(* IEC 61131-3 sources: RECIRS/QEMUv8/OpenPLC_v3/webserver/st_files, 24 files *)

(* ---- 7_segment_display.st ---- *)
PROGRAM prog0

VAR
    Rdosc : BOOL;
    Cdigit : INT;
    digit : INT;
    digit0 : INT;
    digit1 : INT;
    digit2 : INT;

    Ycom_digit0 : BOOL;
    Ycom_digit1 : BOOL;
    Ycom_digit2 : BOOL;
    Yseg_a : BOOL;
    Yseg_b : BOOL;
    Yseg_c : BOOL;
    Yseg_d : BOOL;
    Yseg_e : BOOL;
    Yseg_f : BOOL;
    Yseg_g : BOOL;
END_VAR

Rdosc := FALSE;

IF Rdosc THEN
    Rdosc := TRUE;
END_IF;

IF Rdosc THEN
    Cdigit := Cdigit + 1;
    IF Cdigit > 2 THEN
        Cdigit := 0;
    END_IF;
END_IF;

CASE Cdigit OF
    0:
        Ycom_digit0 := TRUE;
        Ycom_digit1 := FALSE;
        Ycom_digit2 := FALSE;
        digit := digit0;
    1:
        Ycom_digit0 := FALSE;
        Ycom_digit1 := TRUE;
        Ycom_digit2 := FALSE;
        digit := digit1;
    2:
        Ycom_digit0 := FALSE;
        Ycom_digit1 := FALSE;
        Ycom_digit2 := TRUE;
        digit := digit2;
END_CASE;

Yseg_a := (digit <> 1) AND (digit <> 4);
Yseg_b := (digit <> 5) AND (digit <> 6);
Yseg_c := (digit <> 2);
Yseg_d := (digit <> 1) AND (digit <> 4) AND (digit <> 7);
Yseg_e := (digit = 0) OR (digit = 2) OR (digit = 6) OR (digit = 8);
Yseg_f := (digit <> 1) AND (digit <> 2) AND (digit <> 3) AND (digit <> 7);
Yseg_g := (digit <> 0) AND (digit <> 1) AND (digit <> 7);

digit0 := 1;
digit1 := 8;
digit2 := 5;

END_PROGRAM

CONFIGURATION Config0

  RESOURCE Res0 ON PLC
    TASK Main(INTERVAL := T#100ms,PRIORITY := 0);
    PROGRAM Inst0 WITH Main : prog0;
  END_RESOURCE
END_CONFIGURATION

(* ---- blank_program.st ---- *)
PROGRAM prog0
  VAR
    var_in : BOOL;
    var_out : BOOL;
  END_VAR

  var_out := var_in;
END_PROGRAM

CONFIGURATION Config0

  RESOURCE Res0 ON PLC
    TASK Main(INTERVAL := T#1ms,PRIORITY := 0);
    PROGRAM Inst0 WITH Main : prog0;
  END_RESOURCE
END_CONFIGURATION

(* ---- brewing_system.st ---- *)
PROGRAM prog0
VAR
    StartButton : BOOL;
    StopButton : BOOL;
    Brewing : BOOL;
    Heating : BOOL;
    Cooling : BOOL;
    Fermenting : BOOL;
    TimerHeat : TON;
    TimerCool : TON;
    TimerFerment : TON;
    StartTrigger : R_TRIG;
    StopTrigger : F_TRIG;
    TempSetPoint : REAL := 65.0;
    _TEMPCurrent : REAL;
    CurrentTemp : REAL := 20.0;
    TempChangeRate : REAL := 0.5;
END_VAR

IF CurrentTemp < TempSetPoint THEN
	StartButton := TRUE;
END_IF;

StartTrigger(CLK := StartButton);
StopTrigger(CLK := StopButton);

IF StartTrigger.Q THEN
    Brewing := TRUE;
    TimerHeat(IN := TRUE, PT := T#1h);
    Heating := TimerHeat.Q;
    IF TimerHeat.Q THEN
        TimerCool(IN := TRUE, PT := T#30m);
        Cooling := TimerCool.Q;
    END_IF;
    IF TimerCool.Q THEN
        TimerFerment(IN := TRUE, PT := T#7d);
        Fermenting := TimerFerment.Q;
    END_IF;
ELSE
    Brewing := FALSE;
    TimerHeat(IN := FALSE);
    TimerCool(IN := FALSE);
    TimerFerment(IN := FALSE);
    Heating := FALSE;
    Cooling := FALSE;
    Fermenting := FALSE;
END_IF;

IF StopTrigger.Q THEN
    Brewing := FALSE;
    Heating := FALSE;
    Cooling := FALSE;
    Fermenting := FALSE;
END_IF;

IF Heating THEN
	_TEMPCurrent := MUL(TempChangeRate, 0.1);
	CurrentTemp := ADD(CurrentTemp, _TEMPCurrent);
ELSIF Cooling THEN
	_TEMPCurrent := MUL(TempChangeRate, 0.1);
	CurrentTemp := SUB(CurrentTemp, _TEMPCurrent);
END_IF;

END_PROGRAM

CONFIGURATION Config0

  RESOURCE Res0 ON PLC
    TASK Main(INTERVAL := T#50ms,PRIORITY := 0);
    PROGRAM Inst0 WITH Main : prog0;
  END_RESOURCE
END_CONFIGURATION

(* ---- car_wash.st ---- *)
PROGRAM prog0
VAR
    StartButton : BOOL := TRUE;
    StopButton : BOOL;
    CarDetected : BOOL;
    Washing : BOOL;
    Rinsing : BOOL;
    Drying : BOOL;
    TimerWash : TON;
    TimerRinse : TON;
    TimerDry : TON;
    StartTrigger : R_TRIG;
    StopTrigger : F_TRIG;
    _TEMP : REAL;
    CarPosition : REAL := 0.0;
    CarSpeed : REAL := 0.5;
    WashPosition : REAL := 2.0;
    RinsePosition : REAL := 4.0;
    DryPosition : REAL := 6.0;
END_VAR

StartTrigger(CLK := StartButton);
StopTrigger(CLK := StopButton);

IF StartTrigger.Q AND CarDetected THEN
    TimerWash(IN := TRUE, PT := T#2m);
    Washing := TimerWash.Q;
    IF TimerWash.Q THEN
        TimerRinse(IN := TRUE, PT := T#1m);
        Rinsing := TimerRinse.Q;
    END_IF;
    IF TimerRinse.Q THEN
        TimerDry(IN := TRUE, PT := T#1m);
        Drying := TimerDry.Q;
    END_IF;
ELSE
    TimerWash(IN := FALSE);
    TimerRinse(IN := FALSE);
    TimerDry(IN := FALSE);
    Washing := FALSE;
    Rinsing := FALSE;
    Drying := FALSE;
END_IF;

IF StopTrigger.Q THEN
    Washing := FALSE;
    Rinsing := FALSE;
    Drying := FALSE;
END_IF;

_TEMP := MUL(CarSpeed, 0.1);
IF Washing THEN
	CarPosition := ADD(CarPosition, _TEMP);
	IF CarPosition >= WashPosition THEN
		Washing := FALSE;
		Rinsing := TRUE;
	END_IF;
END_IF;

IF Rinsing THEN
	CarPosition := ADD(CarPosition, _TEMP);
	IF CarPosition >= RinsePosition THEN
		Rinsing := FALSE;
		Drying := TRUE;
	END_IF;
END_IF;

IF Drying THEN
	CarPosition := ADD(CarPosition, _TEMP);
	IF CarPosition >= DryPosition THEN
		Drying := FALSE;
	END_IF;
END_IF;

END_PROGRAM

CONFIGURATION Config0

  RESOURCE Res0 ON PLC
    TASK Main(INTERVAL := T#50ms,PRIORITY := 0);
    PROGRAM Inst0 WITH Main : prog0;
  END_RESOURCE
END_CONFIGURATION

(* ---- conveyor_belt.st ---- *)
PROGRAM program0
  VAR
    start_button : BOOL;
    stop_button : BOOL;
    emergency_button : BOOL;
    proximity_sensor : BOOL;
    motor_forward : BOOL;
    motor_reverse : BOOL;
    conveyor_running : BOOL := TRUE;
    entity_present : BOOL := FALSE;
    total_types : INT := 1;
    entity_type : INT;
    count : INT := 1;
    timer : BOOL;
    TON0 : TON;
    TOF0 : TOF;
    _TMP_ADD29_OUT : INT;
    _TMP_EQ31_OUT : BOOL;
    _TMP_BOOL_TO_INT33_OUT : INT;
    _TMP_MUL35_OUT : INT;
    _TMP_SUB37_OUT : INT;
    _TMP_INT_TO_STRING39_OUT : STRING;
  END_VAR

  TON0(IN := NOT(timer), PT := T#10ms);
  TOF0(IN := TON0.Q, PT := T#10ms);
  timer := TOF0.Q;
  IF NOT entity_present AND NOT proximity_sensor AND conveyor_running THEN
    entity_present := FALSE;
  END_IF;
  IF proximity_sensor AND conveyor_running THEN
    entity_present := TRUE;
  END_IF;
  entity_type := total_types;
  IF emergency_button THEN
    motor_forward := FALSE;
  END_IF;
  IF NOT conveyor_running THEN
    motor_forward := FALSE;
  END_IF;
  IF emergency_button THEN
    motor_reverse := FALSE;
  END_IF;
  _TMP_ADD29_OUT := ADD(count, 1);
  count := _TMP_ADD29_OUT;
  IF NOT conveyor_running THEN
    motor_reverse := FALSE;
  END_IF;
  IF emergency_button THEN
    conveyor_running := FALSE;
  END_IF;
  IF emergency_button THEN
    entity_present := FALSE;
  END_IF;
  _TMP_EQ31_OUT := EQ(count, 5);
  _TMP_BOOL_TO_INT33_OUT := BOOL_TO_INT(_TMP_EQ31_OUT);
  _TMP_MUL35_OUT := MUL(_TMP_BOOL_TO_INT33_OUT, 4);
  _TMP_SUB37_OUT := SUB(count, _TMP_MUL35_OUT);
  count := _TMP_SUB37_OUT;
  IF start_button AND NOT emergency_button THEN
    conveyor_running := TRUE;
  END_IF;
  IF stop_button AND NOT emergency_button THEN
    conveyor_running := FALSE;
  END_IF;
  _TMP_INT_TO_STRING39_OUT := INT_TO_STRING(entity_type);
END_PROGRAM

CONFIGURATION Config0

  RESOURCE Res0 ON PLC
    TASK task0(INTERVAL := T#100ms,PRIORITY := 0);
    PROGRAM instance0 WITH task0 : program0;
  END_RESOURCE
END_CONFIGURATION

(* ---- elevator.st ---- *)
PROGRAM program0
  VAR
    floor_buttons : ARRAY [1..5] OF BOOL;
    door_sensor : BOOL;
    motor_up : BOOL;
    motor_down : BOOL;
    open_door : BOOL;
    close_door : BOOL;
    current_floor : INT := 1;
    target_floor : INT := 1;
    door_opened : BOOL := FALSE;
    count : INT := 1;
  END_VAR

  IF NOT door_opened THEN
      FOR count := 1 TO 5 DO
          IF floor_buttons[count] THEN
              target_floor := count;
          END_IF;
      END_FOR;
      IF target_floor > current_floor THEN
          motor_up := TRUE;
      ELSIF target_floor < current_floor THEN
          motor_up := FALSE;
          motor_down := TRUE;
      ELSE
          motor_up := FALSE;
          motor_down := FALSE;
      END_IF;
      IF target_floor = current_floor THEN
          motor_up := FALSE;
          motor_down := FALSE;
          open_door := TRUE;
          door_opened := TRUE;
      END_IF;
  ELSE
      IF NOT door_sensor THEN
          close_door := TRUE;
      ELSE
          close_door := FALSE;
          open_door := FALSE;
          door_opened := FALSE;
          current_floor := target_floor;
      END_IF;
  END_IF;
END_PROGRAM

CONFIGURATION Config0

  RESOURCE Res0 ON PLC
    TASK task0(INTERVAL := T#1ms,PRIORITY := 0);
    PROGRAM instance0 WITH task0 : program0;
  END_RESOURCE
END_CONFIGURATION

(* ---- energy_manage.st ---- *)
PROGRAM prog0
VAR
    PeakHours : BOOL;
    NonPeakHours : BOOL;
    EnergyConsumption : REAL := 0.0;
    MaxConsumption : REAL := 1000.0;
    LoadShedding : BOOL;
    Timer : TON;
    _TEMP : REAL;
    EnergyGeneration : REAL := 500.0;
    EnergyUsage : REAL := 600.0;
END_VAR

IF PeakHours THEN
    IF EnergyConsumption > MaxConsumption THEN
        LoadShedding := TRUE;
        Timer(IN := TRUE, PT := T#30m);
    ELSE
        LoadShedding := FALSE;
        Timer(IN := FALSE);
    END_IF;
ELSE
    LoadShedding := FALSE;
    Timer(IN := FALSE);
END_IF;

IF Timer.Q THEN
	LoadShedding := FALSE;
END_IF;

IF LoadShedding THEN
	_TEMP := MUL(EnergyUsage, 0.1);
	EnergyConsumption := SUB(EnergyConsumption, _TEMP);
ELSE
	_TEMP := MUL(EnergyGeneration, 0.1);
	EnergyConsumption := ADD(EnergyConsumption, _TEMP);
END_IF;

END_PROGRAM

CONFIGURATION Config0

  RESOURCE Res0 ON PLC
    TASK Main(INTERVAL := T#50ms,PRIORITY := 0);
    PROGRAM Inst0 WITH Main : prog0;
  END_RESOURCE
END_CONFIGURATION

(* ---- gate_controller.st ---- *)
PROGRAM Gate_Controller
  VAR
    Start_Loop : BOOL := False;
    one_hour : TIME := T#1h;
    One_Hour_Timer : TON;
    Gate_Open : BOOL := False;
  END_VAR
  VAR_OUTPUT
    Close_Gate_Inst : BOOL := False;
  END_VAR
  VAR_INPUT
    Sensed_Car : BOOL := False;
    Sensed_Car_Inst : BOOL := False;
    Sensed_App : BOOL := False;
    Mobile_Inst : BOOL := False;
    Auth : STRING;
  END_VAR
  VAR
    my_defined_str : STRING := '"1234"';
  END_VAR

  One_Hour_Timer(IN := NOT(Start_Loop), PT := one_hour);

  IF One_Hour_Timer.Q THEN
    IF Gate_Open THEN
      Close_Gate_Inst := True;
      Gate_Open := False;
    END_IF;
  END_IF;

  IF Sensed_App THEN
    IF EQ(Auth, my_defined_str) THEN
      Close_Gate_Inst := XOR(Mobile_Inst, Gate_Open);
      Gate_Open := Mobile_Inst;
    END_IF;
  END_IF;

  IF Sensed_Car THEN
    IF EQ(Auth, my_defined_str) THEN
      Close_Gate_Inst := XOR(Sensed_Car_Inst, Gate_Open);
      Gate_Open := Sensed_Car_Inst;
    END_IF;
  END_IF;

  Start_Loop := One_Hour_Timer.Q;
END_PROGRAM

CONFIGURATION Config0

  RESOURCE Res0 ON PLC
    TASK task0(INTERVAL := T#20ms,PRIORITY := 0);
    PROGRAM instance0 WITH task0 : Gate_Controller;
  END_RESOURCE
END_CONFIGURATION

(* ---- greenhouse_climate_ctrl.st ---- *)
PROGRAM prog0
VAR
    TempSetPoint : REAL := 22.0;
    HumiditySetPoint : REAL := 60.0;
    CurrentTemp : REAL := 20.0;
    CurrentHumidity : REAL := 55.0;
    HeaterOn : BOOL;
    CoolerOn : BOOL;
    HumidifierOn : BOOL;
    DehumidifierOn : BOOL;
    VentilationOn : BOOL;
    PIDTemp : PID;
    PIDHumidity : PID;
    _TEMP_HEAT : REAL;
    _TEMP_HUMID : REAL;
    TempChangeRate : REAL := 0.1;
    HumidityChangeRate : REAL := 0.2;
END_VAR

PIDTemp(KP := 2.0, TR := 0.5, TD := 0.1, SP := TempSetPoint, PV := CurrentTemp);
PIDHumidity(KP := 1.5, TR := 0.3, TD := 0.1, SP := HumiditySetPoint, PV := CurrentHumidity);

IF PIDTemp.XOUT > 0.0 THEN
    HeaterOn := TRUE;
    CoolerOn := FALSE;
ELSE
    HeaterOn := FALSE;
    CoolerOn := TRUE;
END_IF;

IF PIDHumidity.XOUT > 0.0 THEN
    HumidifierOn := TRUE;
    DehumidifierOn := FALSE;
ELSE
    HumidifierOn := FALSE;
    DehumidifierOn := FALSE;
END_IF;

IF (CurrentTemp > TempSetPoint + 2.0) OR (CurrentHumidity > HumiditySetPoint + 10.0) THEN
    VentilationOn := TRUE;
ELSE
    VentilationOn := FALSE;
END_IF;

IF HeaterOn THEN
	_TEMP_HEAT := MUL(TempChangeRate, 0.1);
	CurrentTemp := ADD(CurrentTemp, _TEMP_HEAT);
ELSIF CoolerOn THEN
	_TEMP_HEAT := MUL(TempChangeRate, 0.1);
	CurrentTemp := SUB(CurrentTemp, _TEMP_HEAT);
END_IF;

IF HumidifierOn THEN
	_TEMP_HUMID := MUL(HumidityChangeRate, 0.1);
	CurrentHumidity := ADD(CurrentHumidity, _TEMP_HUMID);
ELSIF DehumidifierOn THEN
	_TEMP_HUMID := MUL(HumidityChangeRate, 0.1);
	CurrentHumidity := SUB(CurrentHumidity, _TEMP_HUMID);
END_IF;

END_PROGRAM

CONFIGURATION Config0

  RESOURCE Res0 ON PLC
    TASK Main(INTERVAL := T#50ms,PRIORITY := 0);
    PROGRAM Inst0 WITH Main : prog0;
  END_RESOURCE
END_CONFIGURATION

(* ---- hvac.st ---- *)
PROGRAM program0
  VAR
    Heater_enable AT %IX0.1 : BOOL;
  END_VAR
  VAR
    Heater_power : REAL := 0.0;
    Heater_prop : REAL := 0.3;
    Heater_delay : TIME := T#1s;
  END_VAR
  VAR
    Cooler_enable AT %IX0.2 : BOOL;
  END_VAR
  VAR
    Cooler_power : REAL := 0.0;
    Cooler_prop : REAL := -0.1;
    Cooler_delay : TIME := T#1s;
    Fan_enable : BOOL;
    Fan_power : REAL := 0.0;
    Fan_prop : REAL := 0.2;
  END_VAR
  VAR_EXTERNAL
    temperature : REAL;
    temperature_setpoint : REAL;
  END_VAR
  VAR
    temperature_devi : REAL := 0.1;
    Temperature_MIN : REAL := 0.0;
    Temperature_MAX : REAL := 100.0;
    inner_temperature : REAL := 19.0;
    outer_temperature : REAL := 19.0;
    inout_temperature_prop : REAL := 0.001;
  END_VAR
  VAR_EXTERNAL
    humidity : REAL;
  END_VAR
  VAR
    inner_humidity : REAL := 0.45;
    outer_humidity : REAL := 0.35;
  END_VAR
  VAR_EXTERNAL
    humidity_setpoint : REAL;
  END_VAR
  VAR
    humidity_devi : REAL := 0.01;
    humidity_MIN : REAL := 0.0;
    humidity_MAX : REAL := 1.0;
    inout_humidity_prop : REAL := 0.001;
  END_VAR
  VAR_EXTERNAL
    PID_enable : BOOL;
    PID1_enable : BOOL;
    PID_out : REAL;
    PID1_out : REAL;
  END_VAR
  VAR
    PID_zero : REAL := 0.0;
    TON0 : TON;
    TON1 : TON;
    _TMP_ADD87_OUT : REAL;
    _TMP_GT84_OUT : BOOL;
    _TMP_SUB90_OUT : REAL;
    _TMP_LT89_OUT : BOOL;
    _TMP_LIMIT52_OUT : REAL;
    _TMP_LIMIT124_OUT : REAL;
    _TMP_GT72_OUT : BOOL;
    _TMP_EQ65_OUT : BOOL;
    _TMP_LT71_OUT : BOOL;
    _TMP_ADD33_OUT : REAL;
    _TMP_LT29_OUT : BOOL;
    _TMP_SUB38_OUT : REAL;
    _TMP_GT35_OUT : BOOL;
    _TMP_AND91_OUT : BOOL;
    _TMP_MUL6_OUT : REAL;
    _TMP_MUL9_OUT : REAL;
    _TMP_GT93_OUT : BOOL;
    _TMP_BOOL_TO_REAL47_OUT : REAL;
    _TMP_MUL48_OUT : REAL;
    _TMP_ADD49_OUT : REAL;
    _TMP_LT73_OUT : BOOL;
    _TMP_BOOL_TO_REAL58_OUT : REAL;
    _TMP_MUL59_OUT : REAL;
    _TMP_SUB61_OUT : REAL;
    _TMP_BOOL_TO_REAL41_OUT : REAL;
    _TMP_MUL17_OUT : REAL;
    _TMP_ADD40_OUT : REAL;
    _TMP_BOOL_TO_REAL12_OUT : REAL;
    _TMP_MUL23_OUT : REAL;
    _TMP_SUB22_OUT : REAL;
    _TMP_GT108_OUT : BOOL;
    _TMP_BOOL_TO_REAL74_OUT : REAL;
    _TMP_MUL94_OUT : REAL;
    _TMP_ADD96_OUT : REAL;
    _TMP_EQ112_OUT : BOOL;
    _TMP_LT105_OUT : BOOL;
    _TMP_BOOL_TO_REAL100_OUT : REAL;
    _TMP_MUL101_OUT : REAL;
    _TMP_SUB102_OUT : REAL;
    _TMP_MUL118_OUT : REAL;
    _TMP_ADD120_OUT : REAL;
    _TMP_SUB139_OUT : REAL;
    _TMP_LT134_OUT : BOOL;
    _TMP_ADD133_OUT : REAL;
    _TMP_GT131_OUT : BOOL;
    _TMP_ADD147_OUT : REAL;
    _TMP_LT143_OUT : BOOL;
    _TMP_SUB151_OUT : REAL;
    _TMP_GT155_OUT : BOOL;
    _TMP_AND152_OUT : BOOL;
  END_VAR

  _TMP_ADD87_OUT := ADD(temperature_setpoint, temperature_devi);
  _TMP_GT84_OUT := GT(temperature, _TMP_ADD87_OUT);
  _TMP_SUB90_OUT := SUB(temperature_setpoint, temperature_devi);
  _TMP_LT89_OUT := LT(temperature, _TMP_SUB90_OUT);
  IF _TMP_GT84_OUT OR _TMP_LT89_OUT THEN
    PID_enable := TRUE; (*set*)
  END_IF;
  _TMP_LIMIT52_OUT := LIMIT(Temperature_MIN, inner_temperature, Temperature_MAX);
  temperature := _TMP_LIMIT52_OUT;
  IF NOT(PID_enable) THEN
    Heater_enable := FALSE; (*reset*)
  END_IF;
  IF NOT(PID_enable) THEN
    Cooler_enable := FALSE; (*reset*)
  END_IF;
  _TMP_LIMIT124_OUT := LIMIT(humidity_MIN, inner_humidity, humidity_MAX);
  humidity := _TMP_LIMIT124_OUT;
  _TMP_GT72_OUT := GT(PID_out, PID_zero);
  IF _TMP_GT72_OUT THEN
    Heater_enable := TRUE; (*set*)
  END_IF;
  _TMP_EQ65_OUT := EQ(PID_out, PID_zero);
  _TMP_LT71_OUT := LT(PID_out, PID_zero);
  IF _TMP_EQ65_OUT OR _TMP_LT71_OUT THEN
    Heater_enable := FALSE; (*reset*)
  END_IF;
  _TMP_ADD33_OUT := ADD(temperature_setpoint, temperature_devi);
  _TMP_LT29_OUT := LT(temperature, _TMP_ADD33_OUT);
  _TMP_SUB38_OUT := SUB(temperature_setpoint, temperature_devi);
  _TMP_GT35_OUT := GT(temperature, _TMP_SUB38_OUT);
  _TMP_AND91_OUT := AND(_TMP_LT29_OUT, _TMP_GT35_OUT);
  IF _TMP_AND91_OUT THEN
    PID_enable := FALSE; (*reset*)
  END_IF;
  IF _TMP_EQ65_OUT OR _TMP_GT72_OUT THEN
    Cooler_enable := FALSE; (*reset*)
  END_IF;
  IF _TMP_LT71_OUT THEN
    Cooler_enable := TRUE; (*set*)
  END_IF;
  _TMP_MUL6_OUT := MUL(PID_out, Heater_prop);
  Heater_power := _TMP_MUL6_OUT;
  _TMP_MUL9_OUT := MUL(PID_out, Cooler_prop);
  Cooler_power := _TMP_MUL9_OUT;
  _TMP_GT93_OUT := GT(outer_temperature, inner_temperature);
  _TMP_BOOL_TO_REAL47_OUT := BOOL_TO_REAL(_TMP_GT93_OUT);
  _TMP_MUL48_OUT := MUL(_TMP_BOOL_TO_REAL47_OUT, inout_temperature_prop);
  _TMP_ADD49_OUT := ADD(_TMP_MUL48_OUT, inner_temperature);
  inner_temperature := _TMP_ADD49_OUT;
  _TMP_LT73_OUT := LT(outer_temperature, inner_temperature);
  _TMP_BOOL_TO_REAL58_OUT := BOOL_TO_REAL(_TMP_LT73_OUT);
  _TMP_MUL59_OUT := MUL(_TMP_BOOL_TO_REAL58_OUT, inout_temperature_prop);
  _TMP_SUB61_OUT := SUB(inner_temperature, _TMP_MUL59_OUT);
  inner_temperature := _TMP_SUB61_OUT;
  TON0(IN := Heater_enable, PT := Heater_delay);
  _TMP_BOOL_TO_REAL41_OUT := BOOL_TO_REAL(TON0.Q);
  _TMP_MUL17_OUT := MUL(_TMP_BOOL_TO_REAL41_OUT, Heater_power);
  _TMP_ADD40_OUT := ADD(_TMP_MUL17_OUT, inner_temperature);
  inner_temperature := _TMP_ADD40_OUT;
  TON1(IN := Cooler_enable, PT := Cooler_delay);
  _TMP_BOOL_TO_REAL12_OUT := BOOL_TO_REAL(TON1.Q);
  _TMP_MUL23_OUT := MUL(_TMP_BOOL_TO_REAL12_OUT, Cooler_power);
  _TMP_SUB22_OUT := SUB(inner_temperature, _TMP_MUL23_OUT);
  inner_temperature := _TMP_SUB22_OUT;
  _TMP_GT108_OUT := GT(outer_humidity, inner_humidity);
  _TMP_BOOL_TO_REAL74_OUT := BOOL_TO_REAL(_TMP_GT108_OUT);
  _TMP_MUL94_OUT := MUL(_TMP_BOOL_TO_REAL74_OUT, inout_humidity_prop);
  _TMP_ADD96_OUT := ADD(_TMP_MUL94_OUT, inner_humidity);
  inner_humidity := _TMP_ADD96_OUT;
  _TMP_EQ112_OUT := EQ(PID1_out, PID_zero);
  IF _TMP_EQ112_OUT THEN
    Fan_enable := FALSE; (*reset*)
  END_IF;
  IF PID1_enable THEN
    Fan_enable := TRUE; (*set*)
  END_IF;
  _TMP_LT105_OUT := LT(outer_humidity, inner_humidity);
  _TMP_BOOL_TO_REAL100_OUT := BOOL_TO_REAL(_TMP_LT105_OUT);
  _TMP_MUL101_OUT := MUL(_TMP_BOOL_TO_REAL100_OUT, inout_humidity_prop);
  _TMP_SUB102_OUT := SUB(inner_humidity, _TMP_MUL101_OUT);
  inner_humidity := _TMP_SUB102_OUT;
  _TMP_MUL118_OUT := MUL(PID1_out, Fan_prop);
  Fan_power := _TMP_MUL118_OUT;
  _TMP_ADD120_OUT := ADD(inner_humidity, Fan_power);
  inner_humidity := _TMP_ADD120_OUT;
  _TMP_SUB139_OUT := SUB(humidity_setpoint, humidity_devi);
  _TMP_LT134_OUT := LT(temperature, _TMP_SUB139_OUT);
  _TMP_ADD133_OUT := ADD(humidity_setpoint, humidity_devi);
  _TMP_GT131_OUT := GT(humidity, _TMP_ADD133_OUT);
  IF _TMP_GT131_OUT OR _TMP_LT134_OUT THEN
    PID1_enable := TRUE; (*set*)
  END_IF;
  _TMP_ADD147_OUT := ADD(humidity_setpoint, humidity_devi);
  _TMP_LT143_OUT := LT(humidity, _TMP_ADD147_OUT);
  _TMP_SUB151_OUT := SUB(humidity_setpoint, humidity_devi);
  _TMP_GT155_OUT := GT(humidity, _TMP_SUB151_OUT);
  _TMP_AND152_OUT := AND(_TMP_LT143_OUT, _TMP_GT155_OUT);
  IF _TMP_AND152_OUT THEN
    PID1_enable := FALSE; (*reset*)
  END_IF;
END_PROGRAM

PROGRAM program1
  VAR
    PID0 : PID;
  END_VAR
  VAR_EXTERNAL
    PID_enable : BOOL;
  END_VAR
  VAR
    PID_X0 : REAL;
    PID_KP : REAL := -0.05;
    PID_TR : REAL := 10.0;
    PID_TD : REAL := 40.0;
    PID_CYCLE : TIME := T#10ms;
  END_VAR
  VAR_EXTERNAL
    temperature : REAL;
    PID_out : REAL;
    temperature_setpoint : REAL;
  END_VAR

  PID0(AUTO := PID_enable, PV := temperature, SP := temperature_setpoint, KP := PID_KP, TR := PID_TR, TD := PID_TD, CYCLE := PID_CYCLE);
  PID_out := PID0.XOUT;
END_PROGRAM

PROGRAM program2
  VAR
    PID1 : PID;
  END_VAR
  VAR_EXTERNAL
    PID1_enable : BOOL;
  END_VAR
  VAR
    PID1_X0 : REAL;
    PID1_KP : REAL := -0.01;
    PID1_TR : REAL := 5.0;
    PID1_TD : REAL := 20.0;
    PID1_CYCLE : TIME := T#10ms;
  END_VAR
  VAR_EXTERNAL
    humidity : REAL;
    PID1_out : REAL;
    humidity_setpoint : REAL;
  END_VAR

  PID1(AUTO := PID1_enable, PV := humidity, SP := humidity_setpoint, KP := PID1_KP, TR := PID1_TR, TD := PID1_TD, CYCLE := PID1_CYCLE);
  PID1_out := PID1.XOUT;
END_PROGRAM

CONFIGURATION Config0

  RESOURCE Res0 ON PLC
    VAR_GLOBAL
      temperature AT %MD0 : REAL := 0.0;
      humidity AT %MD4 : REAL := 0.0;
      PID_out AT %MD8 : REAL := 0.0;
      PID1_out AT %MD12 : REAL := 0.0;
      PID_enable : BOOL := 1;
      PID1_enable : BOOL := 1;
      temperature_setpoint AT %MD16 : REAL := 24.0;
      humidity_setpoint AT %MD20 : REAL := 0.35;
    END_VAR
    TASK task0(INTERVAL := T#10ms,PRIORITY := 0);
    TASK task2(INTERVAL := T#10ms,PRIORITY := 0);
    TASK task1(INTERVAL := T#10ms,PRIORITY := 0);
    PROGRAM instance0 WITH task0 : program0;
    PROGRAM instance2 WITH task2 : program2;
    PROGRAM instance1 WITH task1 : program1;
  END_RESOURCE
END_CONFIGURATION

(* ---- irrigation_system.st ---- *)
PROGRAM prog0
VAR
    SoilMoisture : REAL := 40.0;
    MoistureSetPoint : REAL := 50.0;
    MoistureUpperLimit : REAL := 60.0;
    MoistureLowerLimit : REAL := 30.0;
    IrrigationOn : BOOL;
    IrrigationAddRate : REAL := 5.0;
    Timer : TON;
    MoistureDecayRate : REAL := 0.5;
END_VAR

IF SoilMoisture < MoistureLowerLimit THEN
    IrrigationOn := TRUE;
    Timer(IN := TRUE, PT := T#30m);
ELSE
    IrrigationOn := FALSE;
    Timer(IN := FALSE);
END_IF;

IF Timer.Q THEN
    IrrigationOn := FALSE;
END_IF;

IF IrrigationOn THEN
	SoilMoisture := ADD(SoilMoisture, IrrigationAddRate);
END_IF;

SoilMoisture := SUB(SoilMoisture, MoistureDecayRate);

END_PROGRAM

CONFIGURATION Config0

  RESOURCE Res0 ON PLC
    TASK Main(INTERVAL := T#1s,PRIORITY := 0);
    PROGRAM Inst0 WITH Main : prog0;
  END_RESOURCE
END_CONFIGURATION

(* ---- lighting_system.st ---- *)
PROGRAM prog0
VAR
    MotionDetected : BOOL;
    LightLevel : REAL;
    LightThreshold : REAL := 300.0;
    LightOn : BOOL;
    Timer : TON;
    MotionTrigger : R_TRIG;
    _TEMP : REAL;
    LightDecayRate : REAL := 10.0;
END_VAR

MotionTrigger(CLK := MotionDetected);

IF MotionTrigger.Q THEN
    LightOn := TRUE;
    Timer(IN := TRUE, PT := T#5m);
ELSE
    Timer(IN := FALSE);
END_IF;

IF Timer.Q THEN
    LightOn := FALSE;
END_IF;

IF LightLevel < LightThreshold THEN
    LightOn := TRUE;
ELSE
    LightOn := FALSE;
END_IF;

IF LightOn THEN
	_TEMP := MUL(LightDecayRate, 0.1);
	LightLevel := ADD(LightLevel, _TEMP);
ELSE
	_TEMP := MUL(LightDecayRate, 0.1);
	LightLevel := SUB(LightLevel, _TEMP);
END_IF;

END_PROGRAM

CONFIGURATION Config0

  RESOURCE Res0 ON PLC
    TASK Main(INTERVAL := T#50ms,PRIORITY := 0);
    PROGRAM Inst0 WITH Main : prog0;
  END_RESOURCE
END_CONFIGURATION

(* ---- packaging_system.st ---- *)
PROGRAM prog0
VAR
    StartButton : BOOL := TRUE;
    StopButton : BOOL;
    ConveyorRunning : BOOL;
    PackageDetected : BOOL;
    PackageCount : INT := 0;
    MaxPackages : INT := 100;
    SealerOn : BOOL;
    EjectorOn : BOOL;
    TimerSealer : TON;
    TimerEjector : TON;
    StartTrigger : R_TRIG;
    StopTrigger : F_TRIG;
    ConveyorSpeed : REAL := 1.0;
    ConveyorPosition : REAL := 0.0;
    PackagePositon : REAL := 0.0;
	PackageLength : REAL := 0.5;
	_TEMPPOS : REAL;
END_VAR

StartTrigger(CLK := StartButton);
StopTrigger(CLK := StopButton);

IF StartButton THEN
    ConveyorRunning := TRUE;
ELSIF StopButton THEN
    ConveyorRunning := FALSE;
END_IF;

IF ConveyorRunning THEN
	_TEMPPOS := MUL(ConveyorSpeed, 0.1);
	ConveyorPosition := ADD(ConveyorPosition, _TEMPPOS);
	IF ConveyorPosition >= PackagePositon + PackageLength THEN
		PackageDetected := TRUE;
		PackagePositon := ConveyorPosition;
	ELSE
		PackageDetected := FALSE;
	END_IF;
ELSE
	PackageDetected := FALSE;
END_IF;

IF ConveyorRunning AND PackageDetected THEN
    PackageCount := PackageCount + 1;
    TimerSealer(IN := TRUE, PT := T#5s);
    SealerOn := TimerSealer.Q;
    IF TimerSealer.Q THEN
		TimerEjector(IN := TRUE, PT := T#2s);
		EjectorOn := TimerEjector.Q;
	END_IF;
    IF PackageCount >= MaxPackages THEN
        ConveyorRunning := FALSE;
    END_IF;
ELSE
    TimerSealer(IN := FALSE);
    TimerEjector(IN := FALSE);
    SealerOn := FALSE;
    EjectorOn := FALSE;
END_IF;
END_PROGRAM

CONFIGURATION Config0

  RESOURCE Res0 ON PLC
    TASK Main(INTERVAL := T#50ms,PRIORITY := 0);
    PROGRAM Inst0 WITH Main : prog0;
  END_RESOURCE
END_CONFIGURATION

(* ---- painting_system.st ---- *)
PROGRAM prog0
VAR
    StartButton : BOOL;
    StopButton : BOOL;
    Painting : BOOL;
    PaintLevel : REAL := 0.0;
    PaintThreshold : REAL := 10.0;
    _TEMPPAINT : REAL;
    RefillPaint : BOOL;
    Timer : TON;
    StartTrigger : R_TRIG;
    StopTrigger : F_TRIG;
    PaintUsageRate : REAL := 1.0;
END_VAR

StartTrigger(CLK := StartButton);
StopTrigger(CLK := StopButton);

IF StartTrigger.Q THEN
    Painting := TRUE;
    Timer(IN := TRUE, PT := T#10m);
ELSIF StopTrigger.Q THEN
    Painting := FALSE;
    Timer(IN := FALSE);
END_IF;

IF PaintLevel < PaintThreshold THEN
	StopButton := FALSE;
	StartButton := TRUE;
ELSIF PaintLevel = 100.0 THEN
	StopButton := TRUE;
	StartButton := FALSE;
END_IF;

IF Timer.Q THEN
    Painting := FALSE;
END_IF;

IF Painting THEN
	_TEMPPAINT := MUL(PaintUsageRate, 0.5);
	PaintLevel := ADD(PaintLevel, _TEMPPAINT);
ELSE
	_TEMPPAINT := MUL(PaintUsageRate, 0.1);
	PaintLevel := SUB(PaintLevel, _TEMPPAINT);
END_IF;

END_PROGRAM

CONFIGURATION Config0

  RESOURCE Res0 ON PLC
    TASK Main(INTERVAL := T#50ms,PRIORITY := 0);
    PROGRAM Inst0 WITH Main : prog0;
  END_RESOURCE
END_CONFIGURATION

(* ---- PWM.st ---- *)
PROGRAM program0
  VAR
    level : DINT;
    count : INT := 1;
    input_analog : REAL;
    input_analog_MIN : REAL := 0.0;
    input_analog_MAX : REAL := 3.3;
    input_analog_local : REAL := 0.0;
    _TMP_INT_TO_REAL42_OUT : REAL;
    _TMP_SIN47_OUT : REAL;
    _TMP_ADD48_OUT : REAL;
    _TMP_MUL43_OUT : REAL;
    _TMP_LIMIT35_OUT : INT;
    _TMP_LIMIT31_OUT : REAL;
    _TMP_DIV23_OUT : REAL;
    _TMP_MUL25_OUT : REAL;
    _TMP_REAL_TO_DINT27_OUT : DINT;
    _TMP_EQ29_OUT : BOOL;
    _TMP_BOOL_TO_INT44_OUT : INT;
    _TMP_MUL45_OUT : INT;
    _TMP_SUB46_OUT : INT;
    _TMP_ADD19_OUT : INT;
  END_VAR

  _TMP_INT_TO_REAL42_OUT := INT_TO_REAL(count);
  _TMP_SIN47_OUT := SIN(_TMP_INT_TO_REAL42_OUT);
  _TMP_ADD48_OUT := ADD(_TMP_SIN47_OUT, 1.0);
  _TMP_MUL43_OUT := MUL(_TMP_ADD48_OUT, 1.65);
  input_analog := _TMP_MUL43_OUT;
  _TMP_LIMIT35_OUT := LIMIT(1, count, 200);
  count := _TMP_LIMIT35_OUT;
  _TMP_LIMIT31_OUT := LIMIT(input_analog_MIN, input_analog, input_analog_MAX);
  input_analog_local := _TMP_LIMIT31_OUT;
  _TMP_DIV23_OUT := DIV(input_analog_local, input_analog_MAX);
  _TMP_MUL25_OUT := MUL(_TMP_DIV23_OUT, 65535.0);
  _TMP_REAL_TO_DINT27_OUT := REAL_TO_DINT(_TMP_MUL25_OUT);
  level := _TMP_REAL_TO_DINT27_OUT;
  _TMP_EQ29_OUT := EQ(count, 200);
  _TMP_BOOL_TO_INT44_OUT := BOOL_TO_INT(_TMP_EQ29_OUT);
  _TMP_MUL45_OUT := MUL(_TMP_BOOL_TO_INT44_OUT, 200);
  _TMP_SUB46_OUT := SUB(count, _TMP_MUL45_OUT);
  count := _TMP_SUB46_OUT;
  _TMP_ADD19_OUT := ADD(count, 1);
  count := _TMP_ADD19_OUT;
END_PROGRAM

CONFIGURATION Config0

  RESOURCE Res0 ON PLC
    TASK task0(INTERVAL := T#20ms,PRIORITY := 0);
    PROGRAM instance0 WITH task0 : program0;
  END_RESOURCE
END_CONFIGURATION

(* ---- robot_arm_ctrl.st ---- *)
PROGRAM prog0
VAR
    StartButton : BOOL := TRUE;
    StopButton : BOOL;
    ArmPosition : REAL := 0.0;
    TargetPosition : REAL := 100.0;
    ArmMoving : BOOL;
    ArmSpeed : REAL := 10.0;
    Timer : TON;
    StartTrigger : R_TRIG;
    StopTrigger : F_TRIG;
    ArmAcceleration : REAL := 1.0;
    ArmVelocity : REAL := 0.0;
    _TempArmPosition : REAL;
    _TempTimer : REAL;
END_VAR

StartTrigger(CLK := StartButton);
StopTrigger(CLK := StopButton);

IF StartTrigger.Q THEN
    ArmMoving := TRUE;
    Timer(IN := TRUE, PT := T#10s);
ELSIF StopTrigger.Q THEN
    ArmMoving := FALSE;
    Timer(IN := FALSE);
END_IF;

IF ArmMoving THEN
    IF ArmPosition < TargetPosition THEN
		_TempTimer := TIME_TO_REAL(Timer.ET);
		_TempArmPosition := MUL(ArmSpeed, _TempTimer);
        ArmPosition := ADD(ArmPosition, _TempArmPosition);
    ELSE
        ArmMoving := FALSE;
    END_IF;
END_IF;
END_PROGRAM

CONFIGURATION Config0

  RESOURCE Res0 ON PLC
    TASK Main(INTERVAL := T#50ms,PRIORITY := 0);
    PROGRAM Inst0 WITH Main : prog0;
  END_RESOURCE
END_CONFIGURATION

(* ---- solar_power_manage.st ---- *)
PROGRAM prog0
VAR
    SolarPanelOutput : REAL := 500.0;
    BatteryLevel : REAL := 50.0;
    GridSupply : REAL := 0.0;
    LoadDemand : REAL := 600.0;
    BatteryCharging : BOOL;
    GridSupplyOn : BOOL;
    Timer : TON;
    _TEMP : REAL;
    BatteryDischargeRate : REAL := 10.0;
END_VAR

IF SolarPanelOutput > LoadDemand THEN
    BatteryCharging := TRUE;
    GridSupplyOn := FALSE;
    Timer(IN := TRUE, PT := T#1h);
ELSE
    BatteryCharging := FALSE;
    Timer(IN := FALSE);
    IF BatteryLevel < 20.0 THEN
        GridSupplyOn := TRUE;
    ELSE
        GridSupplyOn := FALSE;
    END_IF;
END_IF;

IF Timer.Q THEN
	BatteryCharging := FALSE;
END_IF;

IF BatteryCharging THEN
	_TEMP := MUL(BatteryDischargeRate, 0.1);
	BatteryLevel := ADD(BatteryLevel, _TEMP);
ELSE
	_TEMP := MUL(BatteryDischargeRate, 0.1);
	BatteryLevel := SUB(BatteryLevel, _TEMP);
END_IF;
END_PROGRAM

CONFIGURATION Config0

  RESOURCE Res0 ON PLC
    TASK Main(INTERVAL := T#50ms,PRIORITY := 0);
    PROGRAM Inst0 WITH Main : prog0;
  END_RESOURCE
END_CONFIGURATION

(* ---- sorting_system.st ---- *)
PROGRAM prog0
VAR
    StartButton : BOOL;
    StopButton : BOOL;
    ConveyorRunning : BOOL;
    ItemDetected : BOOL;
    ItemType : INT;
    SortBin1 : BOOL;
    SortBin2 : BOOL;
    SortBin3 : BOOL;
    Timer : TON;
    StartTrigger : R_TRIG;
    StopTrigger : F_TRIG;
    _TEMPPOS : REAL;
    ConveyorSpeed : REAL := 1.0;
    ConveyorPosition : REAL := 0.0;
    ItemPosition : REAL := 0.0;
    Bin1Position : REAL := 2.0;
    Bin2Position : REAL := 4.0;
    Bin3Position : REAL := 6.0;
END_VAR

StartTrigger(CLK := StartButton);
StopTrigger(CLK := StopButton);

IF StartTrigger.Q THEN
    ConveyorRunning := TRUE;
ELSIF StopTrigger.Q THEN
    ConveyorRunning := FALSE;
END_IF;

IF ConveyorRunning THEN
	_TEMPPOS := MUL(ConveyorSpeed, 0.1);
	ConveyorPosition := ADD(ConveyorPosition, _TEMPPOS);
	IF ConveyorPosition >= ItemPosition + 1.0 THEN
		ItemDetected := TRUE;
		ItemPosition := ConveyorPosition;
	ELSE
		ItemDetected := FALSE;
	END_IF;
ELSE
	ItemDetected := FALSE;
END_IF;

IF ConveyorRunning AND ItemDetected THEN
    CASE ItemType OF
        1:
			SortBin1 := TRUE;
			Timer(IN := TRUE, PT := T#2s);
        2:
			SortBin2 := TRUE;
			Timer(IN := TRUE, PT := T#2s);
        3:
			SortBin3 := TRUE;
			Timer(IN := TRUE, PT := T#2s);
    ELSE
        SortBin1 := FALSE;
        SortBin2 := FALSE;
        SortBin3 := FALSE;
    END_CASE;
END_IF;

IF Timer.Q THEN
	SortBin1 := FALSE;
	SortBin2 := FALSE;
	SortBin3 := FALSE;
END_IF;

END_PROGRAM

CONFIGURATION Config0

  RESOURCE Res0 ON PLC
    TASK Main(INTERVAL := T#50ms,PRIORITY := 0);
    PROGRAM Inst0 WITH Main : prog0;
  END_RESOURCE
END_CONFIGURATION

(* ---- traffic_light.st ---- *)
PROGRAM Trafic_light
  VAR
    TOF0 : TOF;
    Always_True : BOOL := True;
    Delay_PLC_start_up : BOOL;
    TOF1 : TOF;
    TOF2 : TOF;
  END_VAR
  VAR
    O_LEDRed AT %QX100.0 : BOOL;
    O_LEDOrange AT %QX100.1 : BOOL;
    O_LEDGreen AT %QX100.2 : BOOL;
  END_VAR
  VAR
    No_lamps_active_for_1s : BOOL;
    F_TRIG0 : F_TRIG;
    F_TRIG1 : F_TRIG;
    F_TRIG2 : F_TRIG;
    TON0 : TON;
    SR0 : SR;
    TOF3 : TOF;
    TOF4 : TOF;
    TOF5 : TOF;
    _TMP_OR22_OUT : BOOL;
    _TMP_AND29_OUT : BOOL;
    _TMP_AND33_OUT : BOOL;
    _TMP_AND34_OUT : BOOL;
    _TMP_OR13_OUT : BOOL;
    _TMP_NOT14_OUT : BOOL;
  END_VAR

  TON0(IN := Always_True, PT := T#2s);
  SR0(S1 := TON0.Q);
  Delay_PLC_start_up := SR0.Q1;
  F_TRIG2(CLK := O_LEDOrange);
  _TMP_OR22_OUT := OR(No_lamps_active_for_1s, F_TRIG2.Q);
  TOF0(IN := _TMP_OR22_OUT, PT := T#10s);
  _TMP_AND29_OUT := AND(TOF0.Q, Delay_PLC_start_up);
  O_LEDRed := _TMP_AND29_OUT;
  F_TRIG0(CLK := O_LEDGreen);
  TOF1(IN := F_TRIG0.Q, PT := T#4s);
  _TMP_AND33_OUT := AND(TOF1.Q, Delay_PLC_start_up);
  O_LEDOrange := _TMP_AND33_OUT;
  F_TRIG1(CLK := O_LEDRed);
  TOF2(IN := F_TRIG1.Q, PT := T#10s);
  _TMP_AND34_OUT := AND(TOF2.Q, Delay_PLC_start_up);
  O_LEDGreen := _TMP_AND34_OUT;
  TOF3(IN := O_LEDRed, PT := T#1s);
  TOF4(IN := O_LEDGreen, PT := T#1s);
  TOF5(IN := O_LEDOrange, PT := T#1s);
  _TMP_OR13_OUT := OR(TOF3.Q, TOF4.Q, TOF5.Q);
  _TMP_NOT14_OUT := NOT(_TMP_OR13_OUT);
  No_lamps_active_for_1s := _TMP_NOT14_OUT;
END_PROGRAM

CONFIGURATION Config0

  RESOURCE Res0 ON PLC
    TASK task0(INTERVAL := T#20ms,PRIORITY := 0);
    PROGRAM instance0 WITH task0 : Trafic_light;
  END_RESOURCE
END_CONFIGURATION

(* ---- warehouse_system.st ---- *)
PROGRAM prog0
VAR
    StartButton : BOOL := TRUE;
    StopButton : BOOL;
    ConveyorRunning : BOOL;
    ItemDetected : BOOL;
    StorageLocation : INT;
    ArmMoving : BOOL;
    ArmPosition : REAL;
    TargetPosition : REAL := 0.0;
    Timer : TON;
    StartTrigger : R_TRIG;
    StopTrigger : F_TRIG;
    _TEMPPOS : REAL;
    ConveyorSpeed : REAL := 1.0;
    ConveyorPosition : REAL := 0.0;
    ItemPosition : REAL := 0.0;
END_VAR

StartTrigger(CLK := StartButton);
StopTrigger(CLK := StopButton);

IF StartTrigger.Q THEN
    ConveyorRunning := TRUE;
ELSIF StopTrigger.Q THEN
    ConveyorRunning := FALSE;
END_IF;

IF ConveyorRunning THEN
	_TEMPPOS := MUL(ConveyorSpeed, 0.1);
	ConveyorPosition := ADD(ConveyorPosition, _TEMPPOS);
	IF ConveyorPosition >= ItemPosition + 1.0 THEN
		ItemDetected := TRUE;
		ItemPosition := ConveyorPosition;
	ELSE
		ItemDetected := FALSE;
	END_IF;
ELSE
	ItemDetected := FALSE;
END_IF;

IF ConveyorRunning AND ItemDetected THEN
    CASE StorageLocation OF
        1: TargetPosition := 10.0;
        2: TargetPosition := 20.0;
        3: TargetPosition := 30.0;
    ELSE
        TargetPosition := 0.0;
    END_CASE;
    ArmMoving := TRUE;
    Timer(IN := TRUE, PT := T#5s);
END_IF;

IF ArmMoving THEN
    IF ArmPosition < TargetPosition THEN
        ArmPosition := ArmPosition + 1.0;
    ELSE
        ArmMoving := FALSE;
    END_IF;
END_IF;

IF Timer.Q THEN
	ArmMoving := FALSE;
END_IF;

END_PROGRAM

CONFIGURATION Config0

  RESOURCE Res0 ON PLC
    TASK Main(INTERVAL := T#50ms,PRIORITY := 0);
    PROGRAM Inst0 WITH Main : prog0;
  END_RESOURCE
END_CONFIGURATION

(* ---- watertank.st ---- *)
PROGRAM program0
  VAR
    Valve_in : BOOL;
  END_VAR
  VAR_INPUT
    Valve_in_input : BOOL;
  END_VAR
  VAR
    Valve_out : BOOL;
  END_VAR
  VAR_INPUT
    Valve_out_input : BOOL;
  END_VAR
  VAR_EXTERNAL
    water_height : REAL;
  END_VAR
  VAR
    water_heigh_MIN : REAL := 0.0;
    water_height_MAX : REAL := 100.0;
    inner_water_height : REAL := 100.0;
  END_VAR
  VAR_EXTERNAL
    Valve_in_rate : REAL;
  END_VAR
  VAR
    Valve_in_rate_MIN : REAL := 0.0;
    Valve_in_rate_MAX : REAL := 3.0;
    inner_Valve_in_rate : REAL := 0.0;
    Valve_out_rate : REAL := 0.3;
    _TMP_BOOL_TO_REAL41_OUT : REAL;
    _TMP_MUL17_OUT : REAL;
    _TMP_ADD40_OUT : REAL;
    _TMP_BOOL_TO_REAL12_OUT : REAL;
    _TMP_MUL23_OUT : REAL;
    _TMP_SQRT51_OUT : REAL;
    _TMP_MUL27_OUT : REAL;
    _TMP_SUB22_OUT : REAL;
    _TMP_LIMIT52_OUT : REAL;
    _TMP_LIMIT14_OUT : REAL;
  END_VAR

  Valve_in := NOT(Valve_in_input);
  Valve_out := NOT(Valve_out_input);
  _TMP_BOOL_TO_REAL41_OUT := BOOL_TO_REAL(Valve_in);
  _TMP_MUL17_OUT := MUL(_TMP_BOOL_TO_REAL41_OUT, inner_Valve_in_rate);
  _TMP_ADD40_OUT := ADD(_TMP_MUL17_OUT, inner_water_height);
  inner_water_height := _TMP_ADD40_OUT;
  _TMP_BOOL_TO_REAL12_OUT := BOOL_TO_REAL(Valve_out);
  _TMP_MUL23_OUT := MUL(_TMP_BOOL_TO_REAL12_OUT, Valve_out_rate);
  _TMP_SQRT51_OUT := SQRT(inner_water_height);
  _TMP_MUL27_OUT := MUL(_TMP_MUL23_OUT, _TMP_SQRT51_OUT);
  _TMP_SUB22_OUT := SUB(inner_water_height, _TMP_MUL27_OUT);
  inner_water_height := _TMP_SUB22_OUT;
  _TMP_LIMIT52_OUT := LIMIT(water_heigh_MIN, inner_water_height, water_height_MAX);
  water_height := _TMP_LIMIT52_OUT;
  _TMP_LIMIT14_OUT := LIMIT(Valve_in_rate_MIN, Valve_in_rate, Valve_in_rate_MAX);
  inner_Valve_in_rate := _TMP_LIMIT14_OUT;
END_PROGRAM

PROGRAM program1
  VAR
    PID0 : PID;
    PID_Auto : BOOL;
    PID_X0 : REAL := 0.3;
    PID_KP : REAL := -0.3;
    PID_TR : REAL := 1.3;
    PID_TD : REAL := 1.0;
    PID_CYCLE : TIME := T#200ms;
  END_VAR
  VAR_EXTERNAL
    water_height : REAL;
    Valve_in_rate : REAL;
  END_VAR
  VAR_INPUT
    setpoint : REAL := 50.0;
  END_VAR

  PID0(AUTO := NOT(PID_Auto), PV := water_height, SP := setpoint, X0 := PID_X0, KP := PID_KP, TR := PID_TR, TD := PID_TD, CYCLE := PID_CYCLE);
  Valve_in_rate := PID0.XOUT;
END_PROGRAM

CONFIGURATION Config0

  RESOURCE Res0 ON PLC
    VAR_GLOBAL
      water_height : REAL := 100.0;
      Valve_in_rate : REAL := 0.0;
    END_VAR
    TASK task0(INTERVAL := T#200ms,PRIORITY := 0);
    TASK task1(INTERVAL := T#200ms,PRIORITY := 0);
    PROGRAM instance0 WITH task0 : program0;
    PROGRAM instance1 WITH task1 : program1;
  END_RESOURCE
END_CONFIGURATION

(* ---- watertank2.st ---- *)
PROGRAM program0
  VAR
    Valve_1 AT %IX0.1 : BOOL;
    Valve_in_input AT %IX0.0 : BOOL;
    Valve_3 AT %IX0.2 : BOOL;
    Valve_out_input AT %IX0.3 : BOOL;
  END_VAR
  VAR_EXTERNAL
    water_height_1 : REAL;
    water_height_2 : REAL;
  END_VAR
  VAR
    water_heigh_MIN : REAL := 0.0;
    water_height_MAX : REAL := 100.0;
    inner_water_height_1 : REAL := 100.0;
    inner_water_height_2 : REAL := 100.0;
  END_VAR
  VAR_EXTERNAL
    Valve_1_rate : REAL;
  END_VAR
  VAR
    Valve_rate_MIN : REAL := 0.0;
    Valve_rate_MAX : REAL := 3.0;
    inner_Valve_1_rate : REAL := 0.0;
    inner_Valve_2_rate : REAL := 0.1;
    inner_Valve_3_rate : REAL := 0.0;
  END_VAR
  VAR_EXTERNAL
    Valve_3_rate : REAL;
  END_VAR
  VAR
    _TMP_LIMIT52_OUT : REAL;
    _TMP_LIMIT14_OUT : REAL;
    _TMP_BOOL_TO_REAL41_OUT : REAL;
    _TMP_MUL17_OUT : REAL;
    _TMP_ADD40_OUT : REAL;
    _TMP_BOOL_TO_REAL12_OUT : REAL;
    _TMP_MUL23_OUT : REAL;
    _TMP_SQRT51_OUT : REAL;
    _TMP_MUL27_OUT : REAL;
    _TMP_SUB22_OUT : REAL;
    _TMP_LIMIT34_OUT : REAL;
    _TMP_ADD21_OUT : REAL;
    _TMP_LIMIT43_OUT : REAL;
    _TMP_BOOL_TO_REAL63_OUT : REAL;
    _TMP_MUL50_OUT : REAL;
    _TMP_SUB62_OUT : REAL;
  END_VAR

  IF NOT(Valve_in_input) THEN
    Valve_1 := TRUE; (*set*)
  END_IF;
  IF Valve_in_input THEN
    Valve_1 := FALSE; (*reset*)
  END_IF;
  IF NOT(Valve_out_input) THEN
    Valve_3 := TRUE; (*set*)
  END_IF;
  _TMP_LIMIT52_OUT := LIMIT(water_heigh_MIN, inner_water_height_1, water_height_MAX);
  water_height_1 := _TMP_LIMIT52_OUT;
  IF Valve_out_input THEN
    Valve_3 := FALSE; (*reset*)
  END_IF;
  _TMP_LIMIT14_OUT := LIMIT(Valve_rate_MIN, Valve_1_rate, Valve_rate_MAX);
  inner_Valve_1_rate := _TMP_LIMIT14_OUT;
  _TMP_BOOL_TO_REAL41_OUT := BOOL_TO_REAL(Valve_1);
  _TMP_MUL17_OUT := MUL(_TMP_BOOL_TO_REAL41_OUT, inner_Valve_1_rate);
  _TMP_ADD40_OUT := ADD(_TMP_MUL17_OUT, inner_water_height_1);
  inner_water_height_1 := _TMP_ADD40_OUT;
  _TMP_BOOL_TO_REAL12_OUT := BOOL_TO_REAL(TRUE);
  _TMP_MUL23_OUT := MUL(_TMP_BOOL_TO_REAL12_OUT, inner_Valve_2_rate);
  _TMP_SQRT51_OUT := SQRT(inner_water_height_1);
  _TMP_MUL27_OUT := MUL(_TMP_MUL23_OUT, _TMP_SQRT51_OUT);
  _TMP_SUB22_OUT := SUB(inner_water_height_1, _TMP_MUL27_OUT);
  inner_water_height_1 := _TMP_SUB22_OUT;
  _TMP_LIMIT34_OUT := LIMIT(Valve_rate_MIN, Valve_3_rate, Valve_rate_MAX);
  inner_Valve_3_rate := _TMP_LIMIT34_OUT;
  _TMP_ADD21_OUT := ADD(_TMP_MUL27_OUT, inner_water_height_2);
  inner_water_height_2 := _TMP_ADD21_OUT;
  _TMP_LIMIT43_OUT := LIMIT(water_heigh_MIN, inner_water_height_2, water_height_MAX);
  water_height_2 := _TMP_LIMIT43_OUT;
  _TMP_BOOL_TO_REAL63_OUT := BOOL_TO_REAL(Valve_3);
  _TMP_MUL50_OUT := MUL(_TMP_BOOL_TO_REAL63_OUT, inner_Valve_3_rate);
  _TMP_SUB62_OUT := SUB(inner_water_height_2, _TMP_MUL50_OUT);
  inner_water_height_2 := _TMP_SUB62_OUT;
END_PROGRAM

PROGRAM program1
  VAR
    PID1 : PID;
  END_VAR
  VAR
    PID1_Auto AT %IX0.5 : BOOL;
  END_VAR
  VAR
    PID1_X0 : REAL := 0.3;
    PID1_KP : REAL := 0.5;
    PID1_TR : REAL := 1.3;
    PID1_TD : REAL := 1.0;
    PID1_CYCLE : TIME := T#10ms;
  END_VAR
  VAR_EXTERNAL
    water_height_2 : REAL;
    Valve_3_rate : REAL;
  END_VAR
  VAR
    setpoint_2 AT %MD10 : REAL := 30.0;
  END_VAR

  PID1(AUTO := NOT(PID1_Auto), PV := water_height_2, SP := setpoint_2, X0 := PID1_X0, KP := PID1_KP, TR := PID1_TR, TD := PID1_TD, CYCLE := PID1_CYCLE);
  Valve_3_rate := PID1.XOUT;
END_PROGRAM

PROGRAM program2
  VAR
    PID0 : PID;
  END_VAR
  VAR
    PID0_Auto AT %IX0.4 : BOOL;
  END_VAR
  VAR
    PID0_X0 : REAL := 0.3;
    PID0_KP : REAL := -0.3;
    PID0_TR : REAL := 1.3;
    PID0_TD : REAL := 1.0;
    PID0_CYCLE : TIME := T#10ms;
  END_VAR
  VAR_EXTERNAL
    water_height_1 : REAL;
    Valve_1_rate : REAL;
  END_VAR
  VAR
    setpoint_1 AT %MD8 : REAL := 50.0;
  END_VAR

  PID0(AUTO := NOT(PID0_Auto), PV := water_height_1, SP := setpoint_1, X0 := PID0_X0, KP := PID0_KP, TR := PID0_TR, TD := PID0_TD, CYCLE := PID0_CYCLE);
  Valve_1_rate := PID0.XOUT;
END_PROGRAM

CONFIGURATION Config0

  RESOURCE Res0 ON PLC
    VAR_GLOBAL
      water_height_1 AT %MD0 : REAL := 100.0;
      water_height_2 AT %MD1 : REAL := 100.0;
      Valve_1_rate AT %MD4 : REAL := 0.0;
      Valve_3_rate AT %MD5 : REAL := 0.0;
    END_VAR
    TASK task0(INTERVAL := T#200ms,PRIORITY := 0);
    TASK task2(INTERVAL := T#200ms,PRIORITY := 0);
    TASK task1(INTERVAL := T#200ms,PRIORITY := 0);
    PROGRAM instance0 WITH task0 : program0;
    PROGRAM instance2 WITH task2 : program2;
    PROGRAM instance1 WITH task1 : program1;
  END_RESOURCE
END_CONFIGURATION

(* ---- wave_generator.st ---- *)
PROGRAM wave_generator
  VAR
    oscilator : BOOL;
    count_up : BOOL;
    count_down : BOOL;
  END_VAR
  VAR
    output AT %QW0 : UINT;
  END_VAR
  VAR
    TON0 : TON;
    TOF0 : TOF;
    CTUD_UDINT0 : CTUD_UDINT;
    EQ9_OUT : BOOL;
    EQ14_OUT : BOOL;
    R_TRIG1 : R_TRIG;
    R_TRIG2 : R_TRIG;
    UDINT_TO_UINT29_OUT : UINT;
  END_VAR

  TON0(IN := NOT(oscilator), PT := T#1ms);
  TOF0(IN := TON0.Q, PT := T#1ms);
  oscilator := TOF0.Q;
  EQ9_OUT := EQ(output, 0);
  IF EQ9_OUT THEN
    count_up := TRUE; (*set*)
  END_IF;
  IF EQ9_OUT THEN
    count_down := FALSE; (*reset*)
  END_IF;
  EQ14_OUT := EQ(output, 100);
  IF EQ14_OUT THEN
    count_down := TRUE; (*set*)
  END_IF;
  IF EQ14_OUT THEN
    count_up := FALSE; (*reset*)
  END_IF;
  R_TRIG1(CLK := count_up AND oscilator);
  R_TRIG2(CLK := count_down AND oscilator);
  CTUD_UDINT0(CU := R_TRIG1.Q, CD := R_TRIG2.Q, PV := 65536);
  UDINT_TO_UINT29_OUT := UDINT_TO_UINT(CTUD_UDINT0.CV);
  output := UDINT_TO_UINT29_OUT;
END_PROGRAM

CONFIGURATION Config0

  RESOURCE Res0 ON PLC
    TASK task0(INTERVAL := T#100ms,PRIORITY := 0);
    PROGRAM instance0 WITH task0 : wave_generator;
  END_RESOURCE
END_CONFIGURATION

(* ---- webserver_program.st ---- *)
PROGRAM prog0
  VAR
    var_in : BOOL;
    var_out : BOOL;
  END_VAR

  var_out := var_in;
END_PROGRAM

CONFIGURATION Config0

  RESOURCE Res0 ON PLC
    TASK Main(INTERVAL := T#50ms,PRIORITY := 0);
    PROGRAM Inst0 WITH Main : prog0;
  END_RESOURCE
END_CONFIGURATION
